(* CoDeSys 2.3 project: mixing process.pro *)
(* Libraries: STANDARD.LIB 25.11.03 12:18:06, IECSFC.LIB 25.11.03 12:18:06, ANALYZATION.LIB 25.11.03 12:18:06 *)

(* POU PLC_PRG, LD *)
PROGRAM PLC_PRG
VAR
	TIM1: TOF;
	a: TIME;
END_VAR
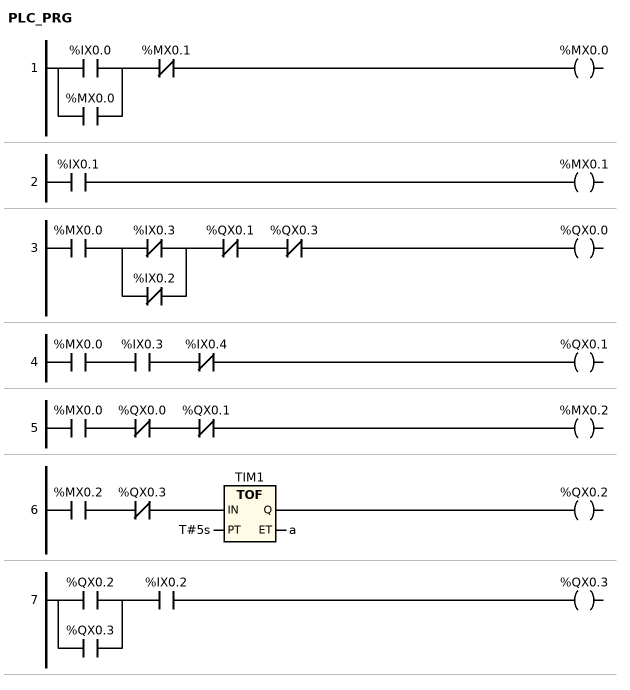
_LD_ (* Ladder Diagram *)
NETWORK 1
	{ [%IX0.0] | [%MX0.0] } - [/%MX0.1] --- (%MX0.0)
NETWORK 2
	[%IX0.1] --- (%MX0.1)
NETWORK 3
	[%MX0.0] - { [/%IX0.3] | [/%IX0.2] } - [/%QX0.1] - [/%QX0.3] --- (%QX0.0)
NETWORK 4
	[%MX0.0] - [%IX0.3] - [/%IX0.4] --- (%QX0.1)
NETWORK 5
	[%MX0.0] - [/%QX0.0] - [/%QX0.1] --- (%MX0.2)
NETWORK 6
	[%MX0.2] - [/%QX0.3] - TIM1:TOF(IN: *, PT: T#5s, ET => a) --- (%QX0.2)
NETWORK 7
	{ [%QX0.2] | [%QX0.3] } - [%IX0.2] --- (%QX0.3)
_END_LD_
(* the same logic as Structured Text *)
(* Network 1 *)
%MX0.0 := (%IX0.0 OR %MX0.0) AND NOT %MX0.1;
(* Network 2 *)
%MX0.1 := %IX0.1;
(* Network 3 *)
%QX0.0 := %MX0.0 AND (NOT %IX0.3 OR NOT %IX0.2) AND NOT %QX0.1 AND NOT %QX0.3;
(* Network 4 *)
%QX0.1 := %MX0.0 AND %IX0.3 AND NOT %IX0.4;
(* Network 5 *)
%MX0.2 := %MX0.0 AND NOT %QX0.0 AND NOT %QX0.1;
(* Network 6 *)
TIM1(IN := %MX0.2 AND NOT %QX0.3, PT := T#5s);
a := TIM1.ET;
%QX0.2 := TIM1.Q;
(* Network 7 *)
%QX0.3 := (%QX0.2 OR %QX0.3) AND %IX0.2;
END_PROGRAM
